// SIMATIC S7-200 SMART project (STEP 7-Micro/WIN SMART), CPU SR40

SYMBOL_TABLE 系统符号
Always_On        SM0.0    // 始终接通
First_Scan_On    SM0.1    // 仅在第一个扫描周期时接通
END_SYMBOL_TABLE

ORGANIZATION_BLOCK MAIN:OB1
TITLE=程序注释
BEGIN
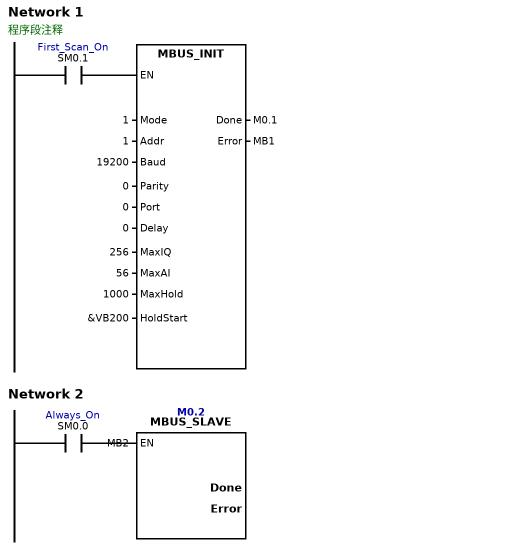
Network 1
// 程序段注释
// (network saved uncompiled; LAD cells follow)
// row 0: c0 -| |- First_Scan_On:SM0.1  c1 [MBUS_INIT EN:=power@row0, Mode:=1, Addr:=1, Baud:=19200, Parity:=0, Port:=0, Delay:=0, MaxIQ:=256, MaxAI:=56, MaxHold:=1000, HoldStart:=&VB200, Done=>M0.1, Error=>MB1]
// row 1: c1 [box]
// row 2: c1 [box]
// row 3: c1 [box]
// row 4: c1 [box]
Network 2
// (network saved uncompiled; LAD cells follow)
// row 0: c0 -| |- Always_On:SM0.0  c1 [MBUS_SLAVE Done Error M0.2 EN:=MB2]
// row 1: c1 [box]
END_ORGANIZATION_BLOCK

// SBR1: protected block, not included

// SBR2: protected block, not included

// SBR3: protected block, not included
